FUNCTION F_ITC_SendGSR : BOOL
(**************************************************************************************
 * 	Application		:	BoxControl Framework
 *	Revision		:	$Revision: 404529 $
 *	Revision date	:	$Date: 2018-04-23 08:21:38 +0200 (Mo., 23 Apr 2018) $
 *	Last changed by	:	$Author: b7bolm $
 *	URL				:	$URL: http://almscdc.swisslog.com/repo/SWPD/Development/BoxControlFramework/20_Release/trunk/01_Software/BCF/BCF/JumpStart/20_Product/10_App/11_Com/10_Lib/10_Conv/11_ITC/F_ITC_SendGSR.TcPOU $
 *
 *	Purpose			:	Wrap message - GSR
 *
 * ------------------------------------------------------------------------------------
 *	Copyright Swisslog [IP AG], Switzerland. All rights reserved.
 * 
 * ------------------------------------------------------------------------------------
 *	
 * 	Revision History: 
 *
 * 	VERSION			DATE			INITIALS			DESCRIPTION
 *	0.1				01.01.2001		swl					Example
 *
 **************************************************************************************)
VAR_INPUT
	eChannelSrc			: E_MFCS_Channel; // Source communicaton channel		
	GroupName			: STRING(Conveyor.POSITION_STRINGLENGTH); // SIS Group Name MM-GGG-0000-000
	eMode				: E_PositionMode; // Mode
	eState				: E_PositionState; // State
	eErrorState			: E_ErrorState; // Error State
	eErrorCode			: E_ErrorConv; // Return Code
	eErrorType			: E_ErrorType; // Error Type
	ErrorInformation	: STRING(System.ERROR_PARAM_STRINGLENGTH); // 5 Chars Error Information
	Variable			: DINT; // Variable
	eReturnCode			: E_ErrorConv; // Return code
END_VAR
VAR
	GSR					: ST_ITC_GSR; 
END_VAR

// Map values
GSR.GroupName := GroupName;
GSR.eState := eState;
GSR.eMode := eMode;
GSR.eErrorCode := eErrorCode;
GSR.eErrorState := eErrorState;
GSR.eErrorType := eErrorType;
GSR.ErrorInformation := ErrorInformation;
GSR.Variable := Variable;
GSR.eReturnCode := eReturnCode;

// Forward to ITC
F_ITC_SendGSR := fbITC_Manager.M_SendData(
					meChannel	:= eChannelSrc,
					mMsgType	:= E_ITC_MsgTypeConv.GROUP_STATUS_REPORT,
					mpData		:= ADR(GSR),
					mLen		:= SIZEOF(GSR));

END_FUNCTION

(* stored: Version 1.1.0.1, ProductVersion 3.1.4022.12
   POU F_ITC_SendGSR: Id {fa16638b-bff5-447f-a388-effaee853e48}, SpecialFunc None *)
